// TIA Portal V17 export
// export: Created 2025-03-13T10:30:24.8016862Z, ExportSetting WithDefaults, DisplayName Totally Integrated Automation Portal, DisplayVersion V17 Update 8, DisplayName TIA Portal Openness, DisplayVersion V17 Update 8, DisplayName TIA Portal Version Control Interface, DisplayVersion V17, DisplayName SINAMICS Startdrive Advanced, DisplayVersion V17 SP2, DisplayName SINAMICS Startdrive G110M, G120, G120C, G120D, G120P, G115D, DisplayVersion V17 SP2, DisplayName SINAMICS Startdrive G130, G150, S120, S150, SINAMICS MV, S210, DisplayVersion V17 SP2, DisplayName STEP 7 Professional, DisplayVersion V17 Update 8, DisplayName SINUMERIK ONE STEP 7 Toolbox, DisplayVersion V17 Update 12, DisplayName SINUMERIK 840D sl STEP 7 Toolbox, DisplayVersion V17 Update 12, DisplayName STEP 7 Safety, DisplayVersion V17 Update 6, DisplayName WinCC Advanced, DisplayVersion V17 Update 8
FUNCTION "FC20201_LASER_TRUMPF_POINTER" : Void   // FC20201, LAD
TITLE = FC20201 LASER TRUMPF POINTER
{ S7_Optimized_Access := 'TRUE' }
VERSION : 0.1
// stored: AutoNumber false, IsIECCheckEnabled false, SetENOAutomatically false, UDAEnableTagReadback false
BEGIN

REGION Network 1: LASER TRUMPF UNIT 1 LASER GUIDE
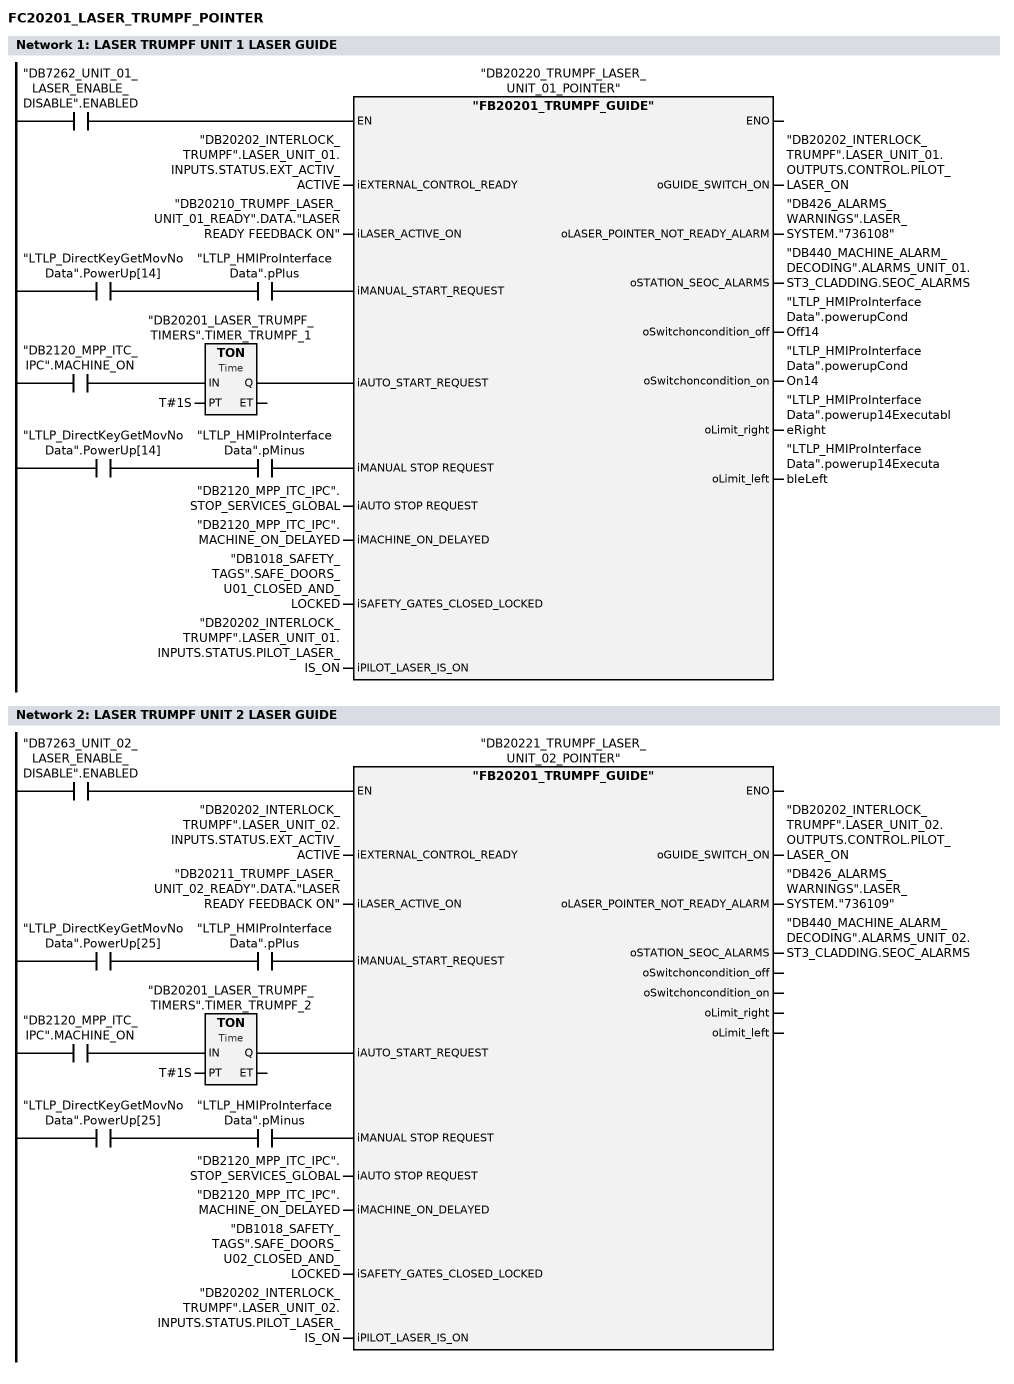
   RUNG wire#powerrail
      Contact( "DB7262_UNIT_01_LASER_ENABLE_DISABLE".ENABLED )
      "DB20220_TRUMPF_LASER_UNIT_01_POINTER"(iMANUAL_START_REQUEST := wire#w1, iAUTO_START_REQUEST := wire#w2, "iMANUAL STOP REQUEST" := wire#w3, iEXTERNAL_CONTROL_READY := "DB20202_INTERLOCK_TRUMPF".LASER_UNIT_01.INPUTS.STATUS.EXT_ACTIV_ACTIVE, iLASER_ACTIVE_ON := "DB20210_TRUMPF_LASER_UNIT_01_READY".DATA."LASER READY FEEDBACK ON", "iAUTO STOP REQUEST" := "DB2120_MPP_ITC_IPC".STOP_SERVICES_GLOBAL, iMACHINE_ON_DELAYED := "DB2120_MPP_ITC_IPC".MACHINE_ON_DELAYED, iSAFETY_GATES_CLOSED_LOCKED := "DB1018_SAFETY_TAGS".SAFE_DOORS_U01_CLOSED_AND_LOCKED, iPILOT_LASER_IS_ON := "DB20202_INTERLOCK_TRUMPF".LASER_UNIT_01.INPUTS.STATUS.PILOT_LASER_IS_ON, oGUIDE_SWITCH_ON => "DB20202_INTERLOCK_TRUMPF".LASER_UNIT_01.OUTPUTS.CONTROL.PILOT_LASER_ON, oLASER_POINTER_NOT_READY_ALARM => "DB426_ALARMS_WARNINGS".LASER_SYSTEM."736108", oSTATION_SEOC_ALARMS => "DB440_MACHINE_ALARM_DECODING".ALARMS_UNIT_01.ST3_CLADDING.SEOC_ALARMS, oSwitchoncondition_off => "LTLP_HMIProInterfaceData".powerupCondOff14, oSwitchoncondition_on => "LTLP_HMIProInterfaceData".powerupCondOn14, oLimit_right => "LTLP_HMIProInterfaceData".powerup14ExecutableRight, oLimit_left => "LTLP_HMIProInterfaceData".powerup14ExecutableLeft)
   END_RUNG
   RUNG wire#powerrail
      Contact( "LTLP_DirectKeyGetMovNoData".PowerUp[14] )
      Contact( "LTLP_HMIProInterfaceData".pPlus )
   END_RUNG wire#w1
   RUNG wire#powerrail
      Contact( "DB2120_MPP_ITC_IPC".MACHINE_ON )
      { S7_Templates := "time_type := Time" } "DB20201_LASER_TRUMPF_TIMERS".TIMER_TRUMPF_1.TON(pt := T#1S, et =>)
   END_RUNG wire#w2
   RUNG wire#powerrail
      Contact( "LTLP_DirectKeyGetMovNoData".PowerUp[14] )
      Contact( "LTLP_HMIProInterfaceData".pMinus )
   END_RUNG wire#w3
   // the same network as SCL:
   "DB20201_LASER_TRUMPF_TIMERS".TIMER_TRUMPF_1.TON(IN := "DB2120_MPP_ITC_IPC".MACHINE_ON, PT := T#1S);
   IF "DB7262_UNIT_01_LASER_ENABLE_DISABLE".ENABLED THEN
       "DB20220_TRUMPF_LASER_UNIT_01_POINTER"(iEXTERNAL_CONTROL_READY := "DB20202_INTERLOCK_TRUMPF".LASER_UNIT_01.INPUTS.STATUS.EXT_ACTIV_ACTIVE,   // "FB20201_TRUMPF_GUIDE"
                               iLASER_ACTIVE_ON := "DB20210_TRUMPF_LASER_UNIT_01_READY".DATA."LASER READY FEEDBACK ON",
                               iMANUAL_START_REQUEST := "LTLP_DirectKeyGetMovNoData".PowerUp[14] AND "LTLP_HMIProInterfaceData".pPlus,
                               iAUTO_START_REQUEST := "DB20201_LASER_TRUMPF_TIMERS".TIMER_TRUMPF_1.Q,
                               "iMANUAL STOP REQUEST" := "LTLP_DirectKeyGetMovNoData".PowerUp[14] AND "LTLP_HMIProInterfaceData".pMinus,
                               "iAUTO STOP REQUEST" := "DB2120_MPP_ITC_IPC".STOP_SERVICES_GLOBAL,
                               iMACHINE_ON_DELAYED := "DB2120_MPP_ITC_IPC".MACHINE_ON_DELAYED,
                               iSAFETY_GATES_CLOSED_LOCKED := "DB1018_SAFETY_TAGS".SAFE_DOORS_U01_CLOSED_AND_LOCKED,
                               iPILOT_LASER_IS_ON := "DB20202_INTERLOCK_TRUMPF".LASER_UNIT_01.INPUTS.STATUS.PILOT_LASER_IS_ON,
                               oGUIDE_SWITCH_ON => "DB20202_INTERLOCK_TRUMPF".LASER_UNIT_01.OUTPUTS.CONTROL.PILOT_LASER_ON,
                               oLASER_POINTER_NOT_READY_ALARM => "DB426_ALARMS_WARNINGS".LASER_SYSTEM."736108",
                               oSTATION_SEOC_ALARMS => "DB440_MACHINE_ALARM_DECODING".ALARMS_UNIT_01.ST3_CLADDING.SEOC_ALARMS,
                               oSwitchoncondition_off => "LTLP_HMIProInterfaceData".powerupCondOff14,
                               oSwitchoncondition_on => "LTLP_HMIProInterfaceData".powerupCondOn14,
                               oLimit_right => "LTLP_HMIProInterfaceData".powerup14ExecutableRight,
                               oLimit_left => "LTLP_HMIProInterfaceData".powerup14ExecutableLeft);
   END_IF;
END_REGION

REGION Network 2: LASER TRUMPF UNIT 2 LASER GUIDE
   RUNG wire#powerrail
      Contact( "DB7263_UNIT_02_LASER_ENABLE_DISABLE".ENABLED )
      "DB20221_TRUMPF_LASER_UNIT_02_POINTER"(iMANUAL_START_REQUEST := wire#w1, iAUTO_START_REQUEST := wire#w2, "iMANUAL STOP REQUEST" := wire#w3, iEXTERNAL_CONTROL_READY := "DB20202_INTERLOCK_TRUMPF".LASER_UNIT_02.INPUTS.STATUS.EXT_ACTIV_ACTIVE, iLASER_ACTIVE_ON := "DB20211_TRUMPF_LASER_UNIT_02_READY".DATA."LASER READY FEEDBACK ON", "iAUTO STOP REQUEST" := "DB2120_MPP_ITC_IPC".STOP_SERVICES_GLOBAL, iMACHINE_ON_DELAYED := "DB2120_MPP_ITC_IPC".MACHINE_ON_DELAYED, iSAFETY_GATES_CLOSED_LOCKED := "DB1018_SAFETY_TAGS".SAFE_DOORS_U02_CLOSED_AND_LOCKED, iPILOT_LASER_IS_ON := "DB20202_INTERLOCK_TRUMPF".LASER_UNIT_02.INPUTS.STATUS.PILOT_LASER_IS_ON, oGUIDE_SWITCH_ON => "DB20202_INTERLOCK_TRUMPF".LASER_UNIT_02.OUTPUTS.CONTROL.PILOT_LASER_ON, oLASER_POINTER_NOT_READY_ALARM => "DB426_ALARMS_WARNINGS".LASER_SYSTEM."736109", oSTATION_SEOC_ALARMS => "DB440_MACHINE_ALARM_DECODING".ALARMS_UNIT_02.ST3_CLADDING.SEOC_ALARMS, oSwitchoncondition_off =>, oSwitchoncondition_on =>, oLimit_right =>, oLimit_left =>)
   END_RUNG
   RUNG wire#powerrail
      Contact( "LTLP_DirectKeyGetMovNoData".PowerUp[25] )
      Contact( "LTLP_HMIProInterfaceData".pPlus )
   END_RUNG wire#w1
   RUNG wire#powerrail
      Contact( "DB2120_MPP_ITC_IPC".MACHINE_ON )
      { S7_Templates := "time_type := Time" } "DB20201_LASER_TRUMPF_TIMERS".TIMER_TRUMPF_2.TON(pt := T#1S, et =>)
   END_RUNG wire#w2
   RUNG wire#powerrail
      Contact( "LTLP_DirectKeyGetMovNoData".PowerUp[25] )
      Contact( "LTLP_HMIProInterfaceData".pMinus )
   END_RUNG wire#w3
   // the same network as SCL:
   "DB20201_LASER_TRUMPF_TIMERS".TIMER_TRUMPF_2.TON(IN := "DB2120_MPP_ITC_IPC".MACHINE_ON, PT := T#1S);
   IF "DB7263_UNIT_02_LASER_ENABLE_DISABLE".ENABLED THEN
       "DB20221_TRUMPF_LASER_UNIT_02_POINTER"(iEXTERNAL_CONTROL_READY := "DB20202_INTERLOCK_TRUMPF".LASER_UNIT_02.INPUTS.STATUS.EXT_ACTIV_ACTIVE,   // "FB20201_TRUMPF_GUIDE"
                               iLASER_ACTIVE_ON := "DB20211_TRUMPF_LASER_UNIT_02_READY".DATA."LASER READY FEEDBACK ON",
                               iMANUAL_START_REQUEST := "LTLP_DirectKeyGetMovNoData".PowerUp[25] AND "LTLP_HMIProInterfaceData".pPlus,
                               iAUTO_START_REQUEST := "DB20201_LASER_TRUMPF_TIMERS".TIMER_TRUMPF_2.Q,
                               "iMANUAL STOP REQUEST" := "LTLP_DirectKeyGetMovNoData".PowerUp[25] AND "LTLP_HMIProInterfaceData".pMinus,
                               "iAUTO STOP REQUEST" := "DB2120_MPP_ITC_IPC".STOP_SERVICES_GLOBAL,
                               iMACHINE_ON_DELAYED := "DB2120_MPP_ITC_IPC".MACHINE_ON_DELAYED,
                               iSAFETY_GATES_CLOSED_LOCKED := "DB1018_SAFETY_TAGS".SAFE_DOORS_U02_CLOSED_AND_LOCKED,
                               iPILOT_LASER_IS_ON := "DB20202_INTERLOCK_TRUMPF".LASER_UNIT_02.INPUTS.STATUS.PILOT_LASER_IS_ON,
                               oGUIDE_SWITCH_ON => "DB20202_INTERLOCK_TRUMPF".LASER_UNIT_02.OUTPUTS.CONTROL.PILOT_LASER_ON,
                               oLASER_POINTER_NOT_READY_ALARM => "DB426_ALARMS_WARNINGS".LASER_SYSTEM."736109",
                               oSTATION_SEOC_ALARMS => "DB440_MACHINE_ALARM_DECODING".ALARMS_UNIT_02.ST3_CLADDING.SEOC_ALARMS);
   END_IF;
END_REGION
END_FUNCTION
